// TIA Portal V21 export
TYPE "LBC_typeMotorStarterInterface"
TITLE = LBC_typeMotorStarterInterface
// Module interface for external systems
   STRUCT
      commands : "LBC_typeMotorStarterCommands";
      monitoring { ExternalWritable := 'False'} : "LBC_typeMotorStarterProcessValues";
      configuration : "LBC_typeMotorStarterConfiguration";
   END_STRUCT;
END_TYPE
